FUNCTION_BLOCK amb_variation (* Basic FB with empty ECC *)
  (* Standard: 61499-2 *)
  (* Version 1.0, 2021-03-22, Lenovo *)
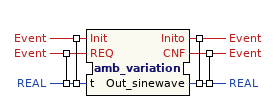
  EVENT_INPUT
    Init WITH t;
    REQ WITH t;
  END_EVENT
  EVENT_OUTPUT
    Inito WITH Out_sinewave;
    CNF WITH Out_sinewave;
  END_EVENT
  VAR_INPUT
    t : REAL;
  END_VAR
  VAR_OUTPUT
    Out_sinewave : REAL;
  END_VAR
  VAR
    freq : REAL; (* Internal Variable *)
    stime : REAL; (* Internal Variable *)
    phase : REAL; (* Internal Variable *)
    f_st : REAL; (* Internal Variable *)
    x : REAL; (* Internal Variable *)
    y : REAL; (* Internal Variable *)
    z : REAL; (* Internal Variable *)
    m : REAL; (* Internal Variable *)
  END_VAR
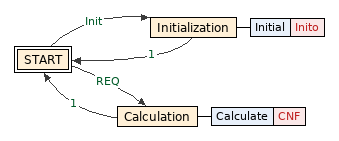
  EC_STATES
    START; (* Initial State *)
    Initialization : Initial -> Inito;
    Calculation : Calculate -> CNF;
  END_STATES
  EC_TRANSITIONS
    START TO Initialization := Init;
    Initialization TO START := 1;
    START TO Calculation := REQ;
    Calculation TO START := 1;
  END_TRANSITIONS
  ALGORITHM Initial IN ST: (* New Algorithm *)

  END_ALGORITHM
  ALGORITHM Calculate IN ST: (* New Algorithm *)
freq:=0.0043633231299859;
phase:=0;
f_st:=freq*t;
x:=f_st+phase;
y:=sin(x);
z:=10*y;;
Out_sinewave:=z;
  END_ALGORITHM
END_FUNCTION_BLOCK
